Yaskawa INFORM job: TT.JBI

/JOB
//NAME TT
///FOLDERNAME FOLDER001
//POS
///NPOS 0,0,0,0,0,0
//INST
///DATE 2025/09/30 17:33
///ATTR SC,RW
///GROUP1 RB1
NOP
*LOOP
WAIT T=0.50
CALL JOB:GO-PARK IF OT#(2393)=ON
CALL JOB:GO-START IF OT#(2394)=ON
CALL JOB:MAKE-UF IF OT#(2395)=ON
CALL JOB:INPUT_WEAVADJ_VALUE IF OT#(2396)=ON
CALL JOB:UPDATE_X_Y_Z IF OT#(2397)=ON
CALL JOB:ABOVE-TO-BELOW IF OT#(2398)=ON
CALL JOB:BELOW-TO-ABOVE IF OT#(2399)=ON
CALL JOB:TEST_ABOVE IF OT#(2400)=ON
CALL JOB:TEST-BELOW IF OT#(2401)=ON
CALL JOB:UPDATE_UF IF OT#(2402)=ON
CALL JOB:GET-BELOW-POSITION IF OT#(2403)=ON
CALL JOB:START-ML IF OT#(2404)=ON
JUMP *LOOP
END
